RoboDK station: RobotCell.rdk

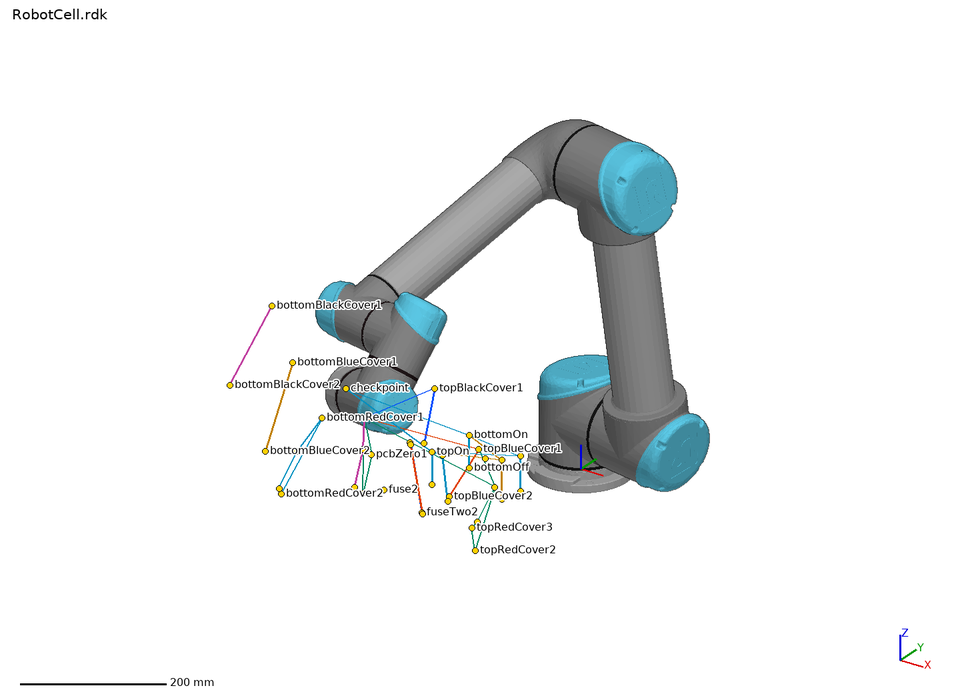
[picture v0: the station drawn from its stored meshes, robots at their saved joint values, targets as dots, program paths as lines]
Station RobotCell2.0 (saved by RoboDK 5.7.0). Poses are relative to the parent item; angles as X-Y-Z fixed-axis rotations.
Station parameters (name, value as stored): IO_0, 0, IO_5, 1, IO_2, 0, IO_1, 0
  - frame UR5 Base at (0, 0, 0) mm
    - robot UR5: 6 axes
        modified DH rows (alpha deg, a mm, theta deg, d mm): 0, 0, 0, 89.2; 90, 0, 180, 0; 0, 425, 0, 0; 0, 392, 0, 109.3; -90, 0, 0, 94.75; 90, 0, 180, 82.5
        joint limits [-360, -360, -360, -360, -360, -360] to [360, 360, 360, 360, 360, 360]; home [0, -90, -90, 0, 90, 0]; saved at [78.868, -81.303, 100.243, -57.656, -163.163, -43.33]
    - target bottomBlueCover2 (Cartesian target) at (-127.51, -571.05, 219.68) mm, rotated rx 155 ry 21.26 rz -138.06 deg; joints [68.539, -66.365, 87.627, -81.498, -103.345, -64.608] of UR5
    - target bottomBlueCover1 (Cartesian target) at (-137.1, -492.19, 320.33) mm, rotated rx 148.39 ry 27.46 rz -138.73 deg; joints [65.104, -77.898, 87.436, -62.46, 251.291, -67.756] of UR5
    - target bottomBlackCover1 (Cartesian target) at (-125.81, -558.63, 435.55) mm, rotated rx 149 ry 27.23 rz -142.77 deg; joints [68.305, -68.522, 57.87, -41.052, 256.19, -61.795] of UR5
    - target bottomBlackCover2 (Cartesian target) at (-125.82, -658.63, 355.55) mm, rotated rx 149 ry 27.23 rz -142.77 deg; joints [71.281, -53.686, 46.921, -44.406, 258.046, -59.407] of UR5
    - target bottomRedCover2 (Cartesian target) at (-131.73, -527.54, 136.12) mm, rotated rx 148.04 ry 26.07 rz -140.48 deg; joints [67.011, -64.579, 98.189, -86.572, -107.302, -64.257] of UR5
    - target bottomRedCover1 (Cartesian target) at (-129.58, -433.27, 214.38) mm, rotated rx 149.87 ry 28.08 rz -142.16 deg; joints [62.435, -81.155, 107.592, -79.242, 253.327, -67.456] of UR5
    - target bottomRedCover3 (Cartesian target) at (-133.02, -530.45, 144.59) mm, rotated rx 148.97 ry 24.46 rz -140.08 deg; joints [67.006, -65.21, 97.856, -87.431, -107.303, -64.271] of UR5
    - target bottomRedCover4 (Cartesian target) at (-137.57, -481.8, 180.64) mm, rotated rx 131.61 ry 42.16 rz -148.61 deg; joints [65.066, -67.661, 95.12, -59.538, 247.973, -63.679] of UR5
    - target pcbTwo1 (Cartesian target) at (28.61, -561.58, 262.06) mm, rotated rx 123.62 ry -1.79 rz -174.84 deg; joints [83.313, -64.127, 76.741, -46.904, -100.825, -5.153] of UR5
    - target pcbTwo2 (Cartesian target) at (28.61, -581.58, 212.06) mm, rotated rx 123.62 ry -1.79 rz -174.84 deg; joints [83.521, -59.604, 77.394, -52.058, -100.653, -5.034] of UR5
    - target pcbZero1 (Cartesian target) at (27.46, -539.77, 244.58) mm, rotated rx 123.08 ry -0.67 rz -177.6 deg; joints [82.574, -66.265, 82.506, -49.742, -98.58, -4.843] of UR5
    - target pcbZero2 (Cartesian target) at (27.46, -559.77, 194.58) mm, rotated rx 123.08 ry -0.67 rz -177.6 deg; joints [82.813, -61.452, 82.987, -55.016, -98.381, -4.71] of UR5
    - target pcb (Cartesian target) at (29.91, -560.04, 309.31) mm, rotated rx 128.13 ry -2.71 rz -175.13 deg; joints [83.404, -66.826, 73.558, -45.608, -100.659, -5.039] of UR5
    - target topBlackCover2 (Cartesian target) at (185.43, -639.82, 346) mm, rotated rx 147.34 ry -27.15 rz 142.81 deg; joints [96.07, -54.236, 48.941, -43.484, -84.83, 49.412] of UR5
    - target topBlackCover1 (Cartesian target) at (184.39, -612.88, 418.75) mm, rotated rx 158.35 ry -16.88 rz 139.06 deg; joints [96.256, -62.574, 52.53, -53.185, -84.989, 49.253] of UR5
    - target topBlueCover2 (Cartesian target) at (187.27, -582.79, 242.47) mm, rotated rx 149.43 ry -30.7 rz 143.31 deg; joints [97.243, -60.964, 74.777, -61.613, -87.92, 51.716] of UR5
    - target topBlueCover1 (Cartesian target) at (180.65, -502.64, 280.78) mm, rotated rx 156.18 ry -24.61 rz 140.55 deg; joints [97.631, -75.075, 89.544, -70.803, -87.916, 51.719] of UR5
    - target topRedCover1 (Cartesian target) at (177.03, -458.86, 205.09) mm, rotated rx 133.52 ry -41.6 rz 154.26 deg; joints [98.03, -70.288, 94.459, -55.176, -88.685, 51.553] of UR5
    - target topRedCover2 (Cartesian target) at (191.26, -526.59, 139.57) mm, rotated rx 142.75 ry -32.65 rz 144.87 deg; joints [97.861, -61.097, 91.158, -72.393, -84.339, 51.767] of UR5
    - target topRedCover3 (Cartesian target) at (193.93, -537.74, 178.7) mm, rotated rx 134.15 ry -38.57 rz 149.99 deg; joints [97.972, -59.569, 82.5, -56.112, -84.309, 51.735] of UR5
    - target topRedCover4 (Cartesian target) at (191.6, -521.43, 181.07) mm, rotated rx 126.33 ry -42.79 rz 155.1 deg; joints [97.966, -59.639, 82.733, -48.998, -84.304, 51.727] of UR5
    - target checkpoint (Cartesian target) at (-62.07, -472.56, 293.21) mm, rotated rx 100.49 ry 5.74 rz -113.36 deg; joints [78.868, -81.303, 100.243, -57.656, -163.163, -43.33] of UR5
    - target topOff (Cartesian target) at (60.78, -442.27, 169.3) mm, rotated rx 91.8 ry -44.65 rz -91.56 deg; joints [94.346, -74.422, 111.459, -52.477, -175.188, 29.272] of UR5
    - target topOn (Cartesian target) at (60.78, -442.27, 219.3) mm, rotated rx 91.8 ry -44.65 rz -91.56 deg; joints [94.346, -78.349, 107.838, -44.93, -175.188, 29.272] of UR5
    - target smash1 (Cartesian target) at (77.78, -442.27, 219.3) mm, rotated rx 91.8 ry -44.65 rz -91.56 deg; joints [96.477, -76.84, 105.632, -39.523, -173.111, 34.006] of UR5
    - target smash2 (Cartesian target) at (79.61, -431.66, 144.82) mm, rotated rx 92.52 ry -47.91 rz -90.3 deg; joints [96.898, -73.248, 114.523, -58.876, -174.407, 30.412] of UR5
    - target bottomOff (Cartesian target) at (76.39, -376.71, 173.1) mm, rotated rx 86.57 ry 44.8 rz -91.72 deg; joints [97.37, -74.248, 111.941, -17.571, -172.906, -24.873] of UR5
    - target bottomOn (Cartesian target) at (76.39, -376.71, 223.1) mm, rotated rx 86.57 ry 44.8 rz -91.72 deg; joints [97.37, -78.255, 108.38, -10.003, -172.906, -24.873] of UR5
    - target clickOn (Cartesian target) at (92.17, -360.2, 185.27) mm, rotated rx 86.58 ry 37.98 rz -90.12 deg; joints [100.078, -76.9, 113.165, -17.794, -171.471, -19.75] of UR5
    - target fuse2 (Cartesian target) at (13.08, -489.09, 167.33) mm, rotated rx 87.33 ry 15.02 rz -178.05 deg; joints [80.669, -58.218, 87.58, -26.723, -101.96, -14.484] of UR5
    - target pcbZeroOff (Cartesian target) at (149.27, -402.92, 156.17) mm, rotated rx 91.21 ry -1.31 rz -87.69 deg; joints [106.419, -71.983, 109.93, -42.891, -165.872, -3.482] of UR5
    - target pcbZeroOn (Cartesian target) at (149.27, -402.91, 216.17) mm, rotated rx 91.21 ry -1.31 rz -87.69 deg; joints [106.419, -76.675, 105.744, -34.012, -165.872, -3.482] of UR5
    - target pcbTwoOff (Cartesian target) at (180.73, -403.22, 177.83) mm, rotated rx 91.25 ry -1.36 rz -87.61 deg; joints [110.153, -71.666, 105.54, -37.969, -162.226, -2.539] of UR5
    - target pcbTwoOn (Cartesian target) at (180.73, -403.22, 230.83) mm, rotated rx 91.25 ry -1.36 rz -87.61 deg; joints [110.153, -75.347, 101.574, -30.323, -162.226, -2.539] of UR5
    - target fuseTwo2 (Cartesian target) at (115.98, -545.45, 184.19) mm, rotated rx 92.33 ry 20.86 rz -173.91 deg; joints [91.297, -52.057, 73.351, -23.48, -93.958, -21.029] of UR5
    - target fuseTwo1 (Cartesian target) at (95.98, -545.45, 284.19) mm, rotated rx 92.33 ry 20.86 rz -173.91 deg; joints [89.473, -56.32, 65.25, -11.122, -95.781, -21.099] of UR5
    - target fuseOne2 (Cartesian target) at (125.2, -557.16, 188.53) mm, rotated rx 93.37 ry 17.82 rz -172.89 deg; joints [92.199, -50.761, 70.226, -22.676, -93.874, -18.062] of UR5
    - target fuseOne1 (Cartesian target) at (105.2, -557.16, 288.54) mm, rotated rx 93.37 ry 17.82 rz -172.89 deg; joints [90.414, -54.707, 61.79, -10.304, -95.657, -18.162] of UR5
  - program setup (3 instructions, listed below)
  - program TopBlack (6 instructions, listed below)
  - program TopBlue (6 instructions, listed below)
  - program TopRed (9 instructions, listed below)
  - program BottomBlack (5 instructions, listed below)
  - program BottomBlue (5 instructions, listed below)
  - program BottomRed (7 instructions, listed below)
  - program FuseOne (3 instructions, listed below)
  - program FuseTwo (3 instructions, listed below)
  - program PCBZero (5 instructions, listed below)
  - program PCBTwo (6 instructions, listed below)
  - program AssembleZero (21 instructions, listed below)
  - program AssembleTwo (33 instructions, listed below)
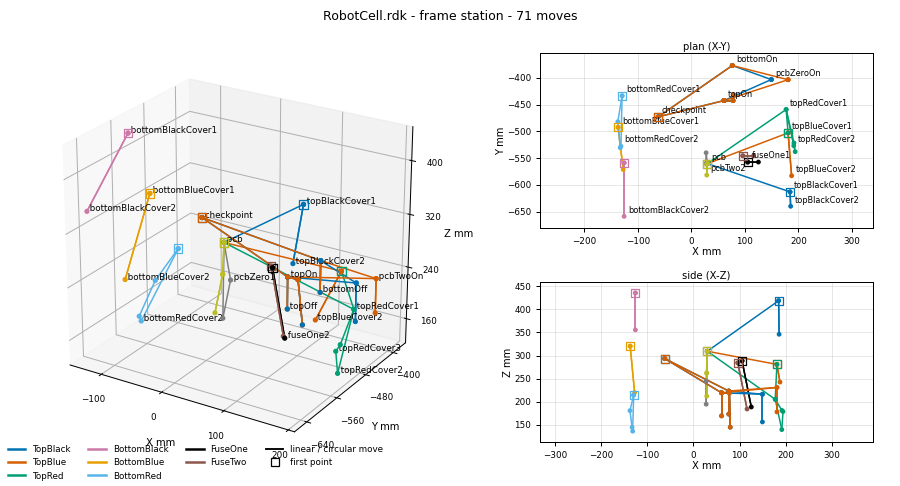
[picture p0: tool path of RobotCell.rdk in frame station, 71 of 71 moves have a stored position in this frame; points joined in program order, loops and branches not executed]

--- program setup (robot UR5) ---
  Set IO_0=0
  Set IO_1=0
  Set IO_2=0

--- program TopBlack (robot UR5) ---
  MoveL (topBlackCover1)
  MoveL (topBlackCover2)
  Set IO_2=1
  Pause 500 ms
  MoveL (topBlackCover1)
  MoveL (pcb)

--- program TopBlue (robot UR5) ---
  MoveL (topBlueCover1)
  MoveL (topBlueCover2)
  Set IO_2=1
  Pause 500 ms
  MoveL (topBlueCover1)
  MoveL (pcb)

--- program TopRed (robot UR5) ---
  MoveL (topBlueCover1)
  MoveL (topRedCover1)
  MoveL (topRedCover2)
  Set IO_2=1
  Pause 500 ms
  MoveL (topRedCover3)
  MoveL (topRedCover4)
  MoveL (topRedCover1)
  MoveL (pcb)

--- program BottomBlack (robot UR5) ---
  MoveL (bottomBlackCover1)
  MoveL (bottomBlackCover2)
  Set IO_0=1
  Pause 500 ms
  MoveL (bottomBlackCover1)

--- program BottomBlue (robot UR5) ---
  MoveL (bottomBlueCover1)
  MoveL (bottomBlueCover2)
  Set IO_0=1
  Pause 500 ms
  MoveL (bottomBlueCover1)

--- program BottomRed (robot UR5) ---
  MoveL (bottomRedCover1)
  MoveL (bottomRedCover2)
  Set IO_0=1
  Pause 500 ms
  MoveL (bottomRedCover3)
  MoveL (bottomRedCover4)
  MoveL (bottomRedCover1)

--- program FuseOne (robot UR5) ---
  MoveL (fuseOne1)
  MoveL (fuseOne2)
  MoveL (fuseOne1)

--- program FuseTwo (robot UR5) ---
  MoveL (fuseTwo1)
  MoveL (fuseTwo2)
  MoveL (fuseTwo1)

--- program PCBZero (robot UR5) ---
  MoveL (pcb)
  MoveL (pcbZero1)
  MoveL (pcbZero2)
  Pause 500 ms
  MoveL (pcb)

--- program PCBTwo (robot UR5) ---
  MoveL (pcb)
  MoveL (pcbTwo1)
  MoveL (pcbTwo2)
  Pause 100 ms
  MoveL (pcbTwo1)
  MoveL (pcb)

--- program AssembleZero (robot UR5) ---
  MoveL (checkpoint)
  MoveL (bottomOn)
  MoveL (bottomOff)
  Set IO_0=0
  MoveL (bottomOn)
  Set IO_0=1
  MoveL (pcbZeroOn)
  Set IO_1=1
  MoveL (pcbZeroOff)
  MoveL (pcbZeroOn)
  Set IO_1=0
  MoveL (topOn)
  MoveL (topOff)
  Set IO_2=0
  MoveL (topOn)
  MoveL (smash1)
  MoveL (smash2)
  MoveL (smash1)
  MoveL (topOn)
  MoveL (checkpoint)
  Set IO_0=0

--- program AssembleTwo (robot UR5) ---
  MoveL (checkpoint)
  MoveL (bottomOn)
  MoveL (bottomOff)
  Set IO_0=0
  MoveL (bottomOn)
  Set IO_0=1
  MoveL (pcbTwoOn)
  MoveL (pcbTwoOff)
  Set IO_1=1
  Pause 100 ms
  Set IO_1=0
  Pause 100 ms
  Set IO_1=1
  Pause 100 ms
  Set IO_1=0
  Pause 100 ms
  Set IO_1=1
  Pause 100 ms
  Set IO_1=0
  Pause 100 ms
  Set IO_1=1
  MoveL (pcbTwoOn)
  Set IO_1=0
  MoveL (topOn)
  MoveL (topOff)
  Set IO_2=0
  MoveL (topOn)
  MoveL (smash1)
  MoveL (smash2)
  MoveL (smash1)
  MoveL (topOn)
  MoveL (checkpoint)
  Set IO_0=0
